{attribute 'qualified_only'}
{attribute 'strict'}
{attribute 'to_string'}
TYPE DUT_CoordSystem :
(
	ACS:=0,
	MCS,
	UCS1,
	UCS2,
	TCP
);
END_TYPE

(* stored: Version 1.1.0.1
   EnumerationTextList DUT_CoordSystem: Id {a6a31ef6-4b82-438e-a7d1-caa766c4a700} *)
